{attribute 'qualified_only'}
{attribute 'strict'}
TYPE E_mode :
(
	default 	:= 0,
	fullmode 	:= 1,
	even 		:= 2,
	odd 		:= 3,
);
END_TYPE

(* stored: Version 1.1.0.1, ProductVersion 3.1.4024.13
   DUT E_mode: Id {1224945f-87b8-4b6f-a2be-5ec4a6b46eb6} *)
